ABB RAPID module: Module1.mod

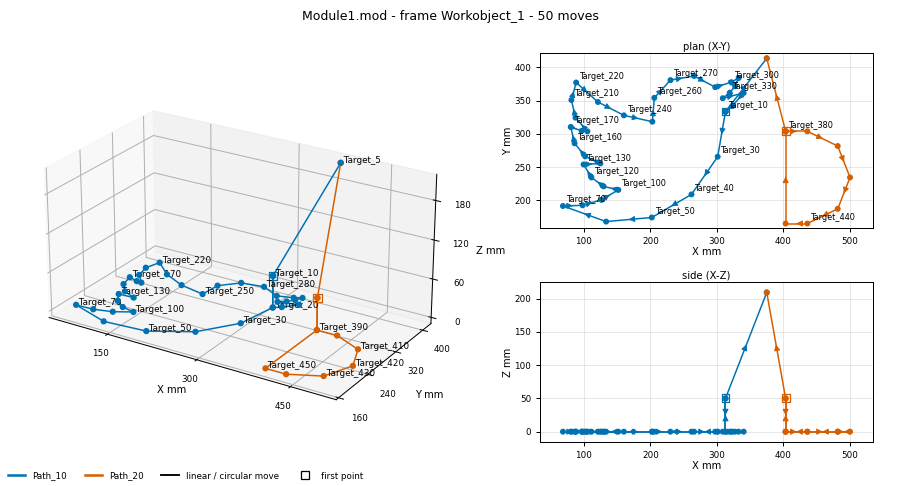
[picture p0: tool path of Module1.mod in frame Workobject_1, 50 of 50 moves have a stored position in this frame; points joined in program order, loops and branches not executed]
MODULE Module1
        CONST robtarget Target_10:=[[312.95280966,333.620099155,50],[0.329310642,0.635971204,-0.606514752,0.34530419],[0,-2,1,0],[9E+09,9E+09,9E+09,9E+09,9E+09,9E+09]];
    CONST robtarget Target_20:=[[312.95280966,333.620099155,0],[0.329310642,0.635971204,-0.606514752,0.34530419],[0,-2,1,0],[9E+09,9E+09,9E+09,9E+09,9E+09,9E+09]];
    CONST robtarget Target_30:=[[301.216986307,265.626968199,0],[0.329310642,0.635971204,-0.606514752,0.34530419],[0,-2,1,0],[9E+09,9E+09,9E+09,9E+09,9E+09,9E+09]];
    CONST robtarget Target_40:=[[261.827524834,208.97658663,0],[0.329310642,0.635971204,-0.606514752,0.34530419],[0,-2,1,0],[9E+09,9E+09,9E+09,9E+09,9E+09,9E+09]];
    CONST robtarget Target_50:=[[202.176009979,174.299617579,0],[0.329310642,0.635971204,-0.606514752,0.34530419],[0,-2,1,0],[9E+09,9E+09,9E+09,9E+09,9E+09,9E+09]];
    CONST robtarget Target_60:=[[133.456279138,168.10332836,0],[0.329310642,0.635971204,-0.606514752,0.34530419],[0,-2,1,0],[9E+09,9E+09,9E+09,9E+09,9E+09,9E+09]];
    CONST robtarget Target_70:=[[68.563855495,191.550476603,0],[0.329310642,0.635971204,-0.606514752,0.34530419],[0,-2,1,0],[9E+09,9E+09,9E+09,9E+09,9E+09,9E+09]];
    CONST robtarget Target_80:=[[98.041612111,192.554722346,0],[0.329310642,0.635971204,-0.606514752,0.34530419],[0,-2,1,0],[9E+09,9E+09,9E+09,9E+09,9E+09,9E+09]];
    CONST robtarget Target_90:=[[126.364950554,200.784858682,0],[0.329310642,0.635971204,-0.606514752,0.34530419],[0,-2,1,0],[9E+09,9E+09,9E+09,9E+09,9E+09,9E+09]];
    CONST robtarget Target_100:=[[151.790538081,215.734311635,0],[0.329310642,0.635971204,-0.606514752,0.34530419],[0,-2,1,0],[9E+09,9E+09,9E+09,9E+09,9E+09,9E+09]];
    CONST robtarget Target_110:=[[129.66038248,221.041225083,0],[0.329310642,0.635971204,-0.606514752,0.34530419],[0,-2,1,0],[9E+09,9E+09,9E+09,9E+09,9E+09,9E+09]];
    CONST robtarget Target_120:=[[111.302142255,234.490467929,0],[0.329310642,0.635971204,-0.606514752,0.34530419],[0,-2,1,0],[9E+09,9E+09,9E+09,9E+09,9E+09,9E+09]];
    CONST robtarget Target_130:=[[99.570180525,253.990934367,0],[0.329310642,0.635971204,-0.606514752,0.34530419],[0,-2,1,0],[9E+09,9E+09,9E+09,9E+09,9E+09,9E+09]];
    CONST robtarget Target_140:=[[124.847619235,255.51629699,0],[0.329310642,0.635971204,-0.606514752,0.34530419],[0,-2,1,0],[9E+09,9E+09,9E+09,9E+09,9E+09,9E+09]];
    CONST robtarget Target_150:=[[101.976138604,266.217877541,0],[0.329310642,0.635971204,-0.606514752,0.34530419],[0,-2,1,0],[9E+09,9E+09,9E+09,9E+09,9E+09,9E+09]];
    CONST robtarget Target_160:=[[86.049407257,285.812970833,0],[0.329310642,0.635971204,-0.606514752,0.34530419],[0,-2,1,0],[9E+09,9E+09,9E+09,9E+09,9E+09,9E+09]];
    CONST robtarget Target_170:=[[80.247736409,310.388752975,0],[0.329310642,0.635971204,-0.606514752,0.34530419],[0,-2,1,0],[9E+09,9E+09,9E+09,9E+09,9E+09,9E+09]];
    CONST robtarget Target_180:=[[96.629366004,304.54518053,0],[0.329310642,0.635971204,-0.606514752,0.34530419],[0,-2,1,0],[9E+09,9E+09,9E+09,9E+09,9E+09,9E+09]];
    CONST robtarget Target_190:=[[105.330574989,303.841706764,0],[0.329310642,0.635971204,-0.606514752,0.34530419],[0,-2,1,0],[9E+09,9E+09,9E+09,9E+09,9E+09,9E+09]];
    CONST robtarget Target_200:=[[87.371126035,324.36364391,0],[0.329310642,0.635971204,-0.606514752,0.34530419],[0,-2,1,0],[9E+09,9E+09,9E+09,9E+09,9E+09,9E+09]];
    CONST robtarget Target_210:=[[81.244437659,350.937228547,0],[0.329310642,0.635971204,-0.606514752,0.34530419],[0,-1,1,0],[9E+09,9E+09,9E+09,9E+09,9E+09,9E+09]];
    CONST robtarget Target_220:=[[88.405679735,377.250881332,0],[0.329310642,0.635971204,-0.606514752,0.34530419],[0,-1,0,0],[9E+09,9E+09,9E+09,9E+09,9E+09,9E+09]];
    CONST robtarget Target_230:=[[121.115546018,347.946582762,0],[0.329310642,0.635971204,-0.606514752,0.34530419],[0,-2,1,0],[9E+09,9E+09,9E+09,9E+09,9E+09,9E+09]];
    CONST robtarget Target_240:=[[160.169714092,327.860537282,0],[0.329310642,0.635971204,-0.606514752,0.34530419],[0,-2,1,0],[9E+09,9E+09,9E+09,9E+09,9E+09,9E+09]];
    CONST robtarget Target_250:=[[203.032450681,318.296904127,0],[0.329310642,0.635971204,-0.606514752,0.34530419],[0,-2,1,0],[9E+09,9E+09,9E+09,9E+09,9E+09,9E+09]];
    CONST robtarget Target_260:=[[205.943517561,354.203728582,0],[0.329310642,0.635971204,-0.606514752,0.34530419],[0,-2,1,0],[9E+09,9E+09,9E+09,9E+09,9E+09,9E+09]];
    CONST robtarget Target_270:=[[230.21652708,380.823183153,0],[0.329310642,0.635971204,-0.606514752,0.34530419],[0,-1,0,0],[9E+09,9E+09,9E+09,9E+09,9E+09,9E+09]];
    CONST robtarget Target_280:=[[265.703151374,387.025912315,0],[0.329310642,0.635971204,-0.606514752,0.34530419],[0,-1,0,0],[9E+09,9E+09,9E+09,9E+09,9E+09,9E+09]];
    CONST robtarget Target_290:=[[297.566750679,370.218610564,0],[0.329310642,0.635971204,-0.606514752,0.34530419],[0,-2,1,0],[9E+09,9E+09,9E+09,9E+09,9E+09,9E+09]];
    CONST robtarget Target_300:=[[321.74298838,377.714052946,0],[0.329310642,0.635971204,-0.606514752,0.34530419],[0,-1,0,0],[9E+09,9E+09,9E+09,9E+09,9E+09,9E+09]];
    CONST robtarget Target_310:=[[332.742941486,384.042138853,0],[0.329310642,0.635971204,-0.606514752,0.34530419],[0,-1,0,0],[9E+09,9E+09,9E+09,9E+09,9E+09,9E+09]];
    CONST robtarget Target_320:=[[327.419478129,372.008881368,0],[0.329310642,0.635971204,-0.606514752,0.34530419],[0,-2,1,0],[9E+09,9E+09,9E+09,9E+09,9E+09,9E+09]];
    CONST robtarget Target_330:=[[319.297487704,361.656499064,0],[0.329310642,0.635971204,-0.606514752,0.34530419],[0,-2,1,0],[9E+09,9E+09,9E+09,9E+09,9E+09,9E+09]];
    CONST robtarget Target_340:=[[308.876898307,353.622206037,0],[0.329310642,0.635971204,-0.606514752,0.34530419],[0,-2,1,0],[9E+09,9E+09,9E+09,9E+09,9E+09,9E+09]];
    CONST robtarget Target_350:=[[340.28609503,361.5363349,0],[0.329310642,0.635971204,-0.606514752,0.34530419],[0,-2,1,0],[9E+09,9E+09,9E+09,9E+09,9E+09,9E+09]];
    CONST robtarget Target_360:=[[323.169462807,341.798469982,0],[0.329310642,0.635971204,-0.606514752,0.34530419],[0,-2,1,0],[9E+09,9E+09,9E+09,9E+09,9E+09,9E+09]];
    CONST robtarget Target_370:=[[312.95280966,333.620099155,0],[0.329310642,0.635971204,-0.606514752,0.34530419],[0,-2,1,0],[9E+09,9E+09,9E+09,9E+09,9E+09,9E+09]];
    CONST robtarget Target_5:=[[375,413.588646413,209.348724977],[0.430459334,0.560985527,-0.560985527,0.430459334],[0,0,0,0],[9E+09,9E+09,9E+09,9E+09,9E+09,9E+09]];
    CONST robtarget Target_380:=[[403.42672598,303.841774112,49.99998461],[0.329310642,0.635971204,-0.606514752,0.34530419],[-1,-1,0,1],[9E+09,9E+09,9E+09,9E+09,9E+09,9E+09]];
    CONST robtarget Target_390:=[[403.426843251,303.841706764,0],[0.329310642,0.635971204,-0.606514752,0.34530419],[-1,-1,0,1],[9E+09,9E+09,9E+09,9E+09,9E+09,9E+09]];
    CONST robtarget Target_400:=[[436.06577659,303.841706764,0],[0.329310642,0.635971204,-0.606514752,0.34530419],[-1,-1,0,1],[9E+09,9E+09,9E+09,9E+09,9E+09,9E+09]];
    CONST robtarget Target_410:=[[481.745763365,281.745155521,0],[0.329310642,0.635971204,-0.606514752,0.34530419],[-1,-1,0,1],[9E+09,9E+09,9E+09,9E+09,9E+09,9E+09]];
    CONST robtarget Target_420:=[[500.257038825,234.498447177,0],[0.329310642,0.635971204,-0.606514752,0.34530419],[-1,-1,0,1],[9E+09,9E+09,9E+09,9E+09,9E+09,9E+09]];
    CONST robtarget Target_430:=[[481.745763365,187.251738833,0],[0.329310642,0.635971204,-0.606514752,0.34530419],[-1,-1,0,1],[9E+09,9E+09,9E+09,9E+09,9E+09,9E+09]];
    CONST robtarget Target_440:=[[436.06577659,165.15518759,0],[0.329310642,0.635971204,-0.606514752,0.34530419],[-1,-1,0,1],[9E+09,9E+09,9E+09,9E+09,9E+09,9E+09]];
    CONST robtarget Target_450:=[[403.426843251,165.15518759,0],[0.329310642,0.635971204,-0.606514752,0.34530419],[-1,-1,0,1],[9E+09,9E+09,9E+09,9E+09,9E+09,9E+09]];
    CONST robtarget Target_460:=[[403.426843251,303.841706764,0],[0.329310642,0.635971204,-0.606514752,0.34530419],[-1,-1,0,1],[9E+09,9E+09,9E+09,9E+09,9E+09,9E+09]];
    CONST robtarget Target_470:=[[403.426843251,303.841706764,50],[0.329310642,0.635971204,-0.606514752,0.34530419],[-1,-1,0,1],[9E+09,9E+09,9E+09,9E+09,9E+09,9E+09]];
!***********************************************************
    !
    ! M?dulo:  Module1
    !
    ! Descripción:
    !   <Introduzca la descripción aquí>
    !
    ! Autor: ASUS
    !
    ! Versión: 1.0
    !
    !***********************************************************


    !***********************************************************
    !
    ! Procedimiento Main
    !
    !   Este es el punto de entrada de su programa
    !
    !***********************************************************
    PROC main()
        Path_10;!Add your code here
    ENDPROC
    PROC Path_10()
        MoveJ Target_10,v600,z10,THerramienta\WObj:=Workobject_1;
        MoveL Target_20,v200,z10,THerramienta\WObj:=Workobject_1;
        MoveL Target_30,v200,z10,THerramienta\WObj:=Workobject_1;
        MoveL Target_40,v200,z10,THerramienta\WObj:=Workobject_1;
        MoveL Target_50,v200,z10,THerramienta\WObj:=Workobject_1;
        MoveL Target_60,v100,z10,THerramienta\WObj:=Workobject_1;
        MoveL Target_70,v100,z10,THerramienta\WObj:=Workobject_1;
        MoveL Target_80,v100,z10,THerramienta\WObj:=Workobject_1;
        MoveL Target_90,v100,z10,THerramienta\WObj:=Workobject_1;
        MoveL Target_100,v100,z10,THerramienta\WObj:=Workobject_1;
        MoveL Target_110,v100,z10,THerramienta\WObj:=Workobject_1;
        MoveL Target_120,v100,z10,THerramienta\WObj:=Workobject_1;
        MoveL Target_130,v100,z10,THerramienta\WObj:=Workobject_1;
        MoveL Target_140,v100,z10,THerramienta\WObj:=Workobject_1;
        MoveL Target_150,v100,z10,THerramienta\WObj:=Workobject_1;
        MoveL Target_160,v100,z10,THerramienta\WObj:=Workobject_1;
        MoveL Target_170,v100,z10,THerramienta\WObj:=Workobject_1;
        MoveL Target_180,v100,z10,THerramienta\WObj:=Workobject_1;
        MoveL Target_190,v100,z10,THerramienta\WObj:=Workobject_1;
        MoveL Target_200,v100,z10,THerramienta\WObj:=Workobject_1;
        MoveL Target_210,v100,z10,THerramienta\WObj:=Workobject_1;
        MoveL Target_220,v100,z10,THerramienta\WObj:=Workobject_1;
        MoveL Target_230,v100,z10,THerramienta\WObj:=Workobject_1;
        MoveL Target_240,v200,z10,THerramienta\WObj:=Workobject_1;
        MoveL Target_250,v200,z10,THerramienta\WObj:=Workobject_1;
        MoveL Target_260,v200,z10,THerramienta\WObj:=Workobject_1;
        MoveL Target_270,v200,z10,THerramienta\WObj:=Workobject_1;
        MoveL Target_280,v400,z10,THerramienta\WObj:=Workobject_1;
        MoveL Target_290,v400,z10,THerramienta\WObj:=Workobject_1;
        MoveL Target_300,v100,z10,THerramienta\WObj:=Workobject_1;
        MoveL Target_310,v100,z10,THerramienta\WObj:=Workobject_1;
        MoveL Target_320,v100,z10,THerramienta\WObj:=Workobject_1;
        MoveL Target_330,v100,z10,THerramienta\WObj:=Workobject_1;
        MoveL Target_340,v100,z10,THerramienta\WObj:=Workobject_1;
        MoveL Target_350,v100,z10,THerramienta\WObj:=Workobject_1;
        MoveL Target_360,v100,z10,THerramienta\WObj:=Workobject_1;
        MoveL Target_370,v100,z10,THerramienta\WObj:=Workobject_1;
        MoveL Target_10,v1000,z100,THerramienta\WObj:=Workobject_1;
        MoveL Target_5,v1000,z100,THerramienta\WObj:=Workobject_1;
    ENDPROC
    PROC first()
        Path_10;
        Path_20;
    ENDPROC
    PROC Path_20()
        MoveL Target_380,v1000,z100,THerramienta\WObj:=Workobject_1;
        MoveL Target_390,v1000,z100,THerramienta\WObj:=Workobject_1;
        MoveL Target_400,v1000,z100,THerramienta\WObj:=Workobject_1;
        MoveL Target_410,v1000,z100,THerramienta\WObj:=Workobject_1;
        MoveL Target_420,v1000,z100,THerramienta\WObj:=Workobject_1;
        MoveL Target_430,v1000,z100,THerramienta\WObj:=Workobject_1;
        MoveL Target_440,v1000,z100,THerramienta\WObj:=Workobject_1;
        MoveL Target_450,v1000,z100,THerramienta\WObj:=Workobject_1;
        MoveL Target_460,v1000,z100,THerramienta\WObj:=Workobject_1;
        MoveL Target_470,v1000,z100,THerramienta\WObj:=Workobject_1;
        MoveL Target_5,v1000,z100,THerramienta\WObj:=Workobject_1;
    ENDPROC
ENDMODULE
